{attribute addProperty BoxType "EL9210-0000-0016"}
{attribute addProperty Id "PowerOKAT %I*PowerOK_5B5BD03A810FuseErrorAT %I*FuseError_3E6D53D3810WcStateAT %I*WcState_F855686C1620InfoDataAT %I*InfoData_192954DE1620"}
{attribute addProperty CRC "2974269189"}
{attribute addProperty SizeInBites "48"}
{attribute addProperty SizeInBytes "6"}
TYPE EL9210_F97BC8F0 :
STRUCT
	{attribute addProperty Name "PowerOK"}
	PowerOK : PowerOK_5B5BD03A;
	{attribute addProperty Name "FuseError"}
	FuseError : FuseError_3E6D53D3;
	{attribute addProperty Name "WcState"}
	WcState : WcState_F855686C;
	{attribute addProperty Name "InfoData"}
	InfoData : InfoData_192954DE;
END_STRUCT
END_TYPE

(* stored: Version 1.2.0.0, ProductVersion 3.1.4024.9
   DUT EL9210_F97BC8F0: Id {45df6370-a7c8-4f2e-83cf-c3e9918bf9af} *)
